FUNCTION_BLOCK FB_Real2Bool_WithParameter (* Basic FB with empty ECC *)
  (* Standard: 61499-2 *)
  (* Version 1.0, 2023-02-20, AK125171 *)
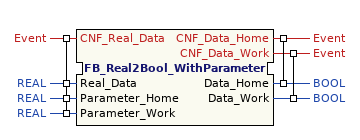
  EVENT_INPUT
    CNF_Real_Data WITH Real_Data, Parameter_Home, Parameter_Work;
  END_EVENT
  EVENT_OUTPUT
    CNF_Data_Home WITH Data_Home; (* IF Real Data is less than 1 *)
    CNF_Data_Work WITH Data_Work; (* If Real Data is more than 9 *)
  END_EVENT
  VAR_INPUT
    Real_Data : REAL;
    Parameter_Home : REAL;
    Parameter_Work : REAL;
  END_VAR
  VAR_OUTPUT
    Data_Home : BOOL;
    Data_Work : BOOL;
  END_VAR
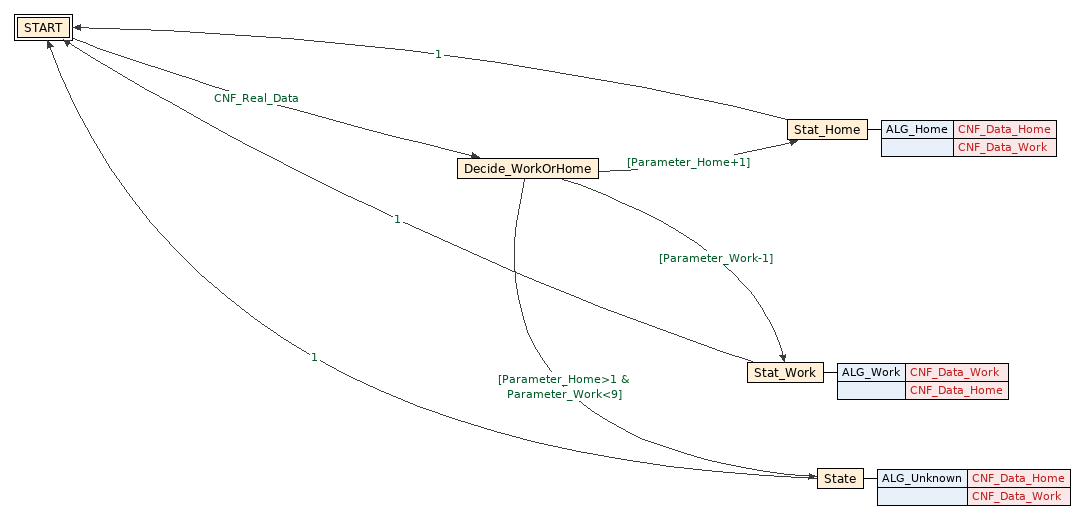
  EC_STATES
    START; (* Initial State *)
    Decide_WorkOrHome;
    Stat_Home : ALG_Home -> CNF_Data_Home, -> CNF_Data_Work;
    Stat_Work : ALG_Work -> CNF_Data_Work, -> CNF_Data_Home;
    State : ALG_Unknown -> CNF_Data_Home, -> CNF_Data_Work;
  END_STATES
  EC_TRANSITIONS
    START TO Decide_WorkOrHome := CNF_Real_Data;
    Decide_WorkOrHome TO Stat_Home := [Parameter_Home+1];
    Decide_WorkOrHome TO Stat_Work := [Parameter_Work-1];
    Stat_Home TO START := 1;
    Stat_Work TO START := 1;
    Decide_WorkOrHome TO State := [Parameter_Home>1 & Parameter_Work<9];
    State TO START := 1;
  END_TRANSITIONS
  ALGORITHM ALG_Work IN ST:
Data_Work:=TRUE;
Data_Home:=FALSE;
  END_ALGORITHM
  ALGORITHM ALG_Home IN ST:
Data_Home:=TRUE;
Data_Work:=FALSE;
  END_ALGORITHM
  ALGORITHM ALG_Unknown IN ST:
Data_Home:=FALSE;
Data_Work:=FALSE;
  END_ALGORITHM
END_FUNCTION_BLOCK
